// TwinCAT 3 PLC project Untitled1
// ProgramVersion: 3.1.4020.2
// libraries:
//   Tc2_Database, * (Beckhoff Automation GmbH)
//   Tc2_Standard, * (Beckhoff Automation GmbH)
//   Tc2_System, * (Beckhoff Automation GmbH)
//   Tc2_Utilities, * (Beckhoff Automation GmbH)
//   Tc3_Module, * (Beckhoff Automation GmbH)
// project tree:
//   DUTs/ ST_Record.TcDUT
//   GVLs/ GVL.TcGVL
//   / PlcTask.TcTTO
//   POUs/ CheckConnection.TcPOU, DatabaseRecord.TcPOU, DatabaseRetrieve.TcPOU, MAIN.TcPOU
// real-time tasks:
//   TASK PlcTask: cycle T#5ms, priority 20, ADS port 350

CONFIGURATION Untitled1
    RESOURCE PLC ON TwinCAT3
        TASK PlcTask(INTERVAL := T#10ms, PRIORITY := 20);
        PROGRAM MAIN WITH PlcTask : MAIN;
    END_RESOURCE
END_CONFIGURATION

// ---- DUTs/ST_Record.TcDUT
TYPE ST_Record :
STRUCT
	ID: T_ULARGE_INTEGER;
	Timestamp: DT;
	temp1: LREAL;
	temp2: LREAL;
	temp3: LREAL;
	bTest: BYTE;
	sComment: STRING;
END_STRUCT
END_TYPE

// ---- GVLs/GVL.TcGVL

VAR_GLOBAL
	(*------ Variable in the database ------*)
	rTemp1 : REAL;
	rTemp2 : REAL;
	rTemp3 : REAL;
	bToggle : INT;
	sComment: STRING;
	
	tStoreVar : TIME := T#5000MS;
	tRetrieveVar: TIME := T#5000MS;
	stRecord : ST_Record;
	nID: T_ULARGE_INTEGER;
END_VAR

// ---- POUs/MAIN.TcPOU
PROGRAM MAIN
VAR
	randomize : DRAND;
	

END_VAR

(*------ Give random values for temperature ------*)
randomize(Seed:= 1, Num=> );
rTemp1 := randomize.Num * 100;
randomize(Seed:= 1, Num=> );
rTemp2 := randomize.Num * 100;
randomize(Seed:= 1, Num=> );
rTemp3 := randomize.Num * 100;

CheckConnection();
DatabaseRecord();
DatabaseRetrieve();

END_PROGRAM

// ---- POUs/CheckConnection.TcPOU
PROGRAM CheckConnection
VAR
	bInit: BOOL := TRUE;
	fbDBOpen : FB_DBConnectionOpen;
	trigger : R_TRIG;
END_VAR

IF bInit THEN
	fbDBOpen(
		hDBID:= 1, 
		bExecute:= TRUE, 
		tTimeout:= T#5S);
	
	(*------ Throw error if there's any ------*)
	trigger(CLK:= fbDBOpen.bError, Q=> );
	IF trigger.Q THEN
		ADSLOGDINT(msgCtrlMask:= ADSLOG_MSGTYPE_MSGBOX, msgFmtStr:= 'Error connecting to database with error ID: %d', dintArg:=fbDBOpen.nErrID );
		RETURN;
	END_IF
	
	(*------ Continue if there's no problem ------*)
	IF NOT fbDBOpen.bBusy AND NOT fbDBOpen.bError THEN
		fbDBOpen.bExecute := FALSE;
		ADSLOGSTR(msgCtrlMask:= ADSLOG_MSGTYPE_LOG, msgFmtStr:= 'Database connection is good', strArg:= '');
		bInit := FALSE;
	END_IF
END_IF

END_PROGRAM

// ---- POUs/DatabaseRecord.TcPOU
PROGRAM DatabaseRecord
VAR
	tTimeout: TIME := T#5s;
	bExecute: BOOL;
	nState: INT;
	
	fbFormatString: FB_FormatString;
	fbDBRecordSelect: FB_DBRecordArraySelect;
	
	timer: TON := (IN:= TRUE);
END_VAR

(*------ Add data to database every tStoreVar time ------*)
timer(IN:= , PT:= tStoreVar, Q=> , ET=> );

fbDBRecordSelect(
	sNetID:= , 
	hDBID:= 1, 
	pCmdAddr:= , 
	cbCmdSize:= , 
	nStartIndex:= 0, 
	nRecordCount:= 1, 
	pDestAddr:= ADR(nID), 
	cbRecordArraySize:= SIZEOF(nID), 
	bExecute:= , 
	tTimeout:= tTimeout);

fbFormatString(
		sFormat:= 'INSERT INTO [myTable] ([Timestamp],[Temperature1],[Temperature2],[Temperature3], [Status], [Comment]) OUTPUT INSERTED.ID VALUES(CURRENT_TIMESTAMP,%0.5f,%0.5f,%0.5f,%d,$'%s$');',  
		arg1:= F_REAL(rTemp1),
		arg2:= F_REAL(rTemp2),
		arg3:= F_REAL(rTemp3),
		arg4:= F_INT(bToggle),
		arg5:= F_STRING(sComment));
(*
//FORMAT FOR MYSQL 
fbFormatString(
		sFormat:= 'INSERT INTO myTable (Timestamp,Temperature1,Temperature2,Temperature3, Status, Comment) VALUES(CURRENT_TIMESTAMP,%0.5f,%0.5f,%0.5f,%d,$'%s$'); SELECT LAST_INSERT_ID();',  
		arg1:= F_REAL(rTemp1),
		arg2:= F_REAL(rTemp2),
		arg3:= F_REAL(rTemp3),
		arg4:= F_INT(bToggle),
		arg5:= F_STRING(sComment));
*)

(*
//FORMAT FOR SQLite 
fbFormatString(
		sFormat:= 'INSERT INTO [myTable] ([Timestamp],[Temperature1],[Temperature2],[Temperature3], [Status], [Comment]) VALUES(CURRENT_TIMESTAMP,%0.5f,%0.5f,%0.5f,%d,$'%s$'); SELECT LAST_INSERT_ROWID();',  
		arg1:= F_REAL(rTemp1),
		arg2:= F_REAL(rTemp2),
		arg3:= F_REAL(rTemp3),
		arg4:= F_INT(bToggle),
		arg5:= F_STRING(sComment));
*)

CASE nState OF 
	0:
	IF NOT fbFormatString.bError AND fbFormatString.sOut <> '' THEN
		nState := 10;
	END_IF

	10:
	IF timer.Q THEN
		fbDBRecordSelect.pCmdAddr := ADR(fbFormatString.sOut);
		fbDBRecordSelect.cbCmdSize := SIZEOF(fbFormatString.sOut);
		fbDBRecordSelect.bExecute := TRUE;
		timer.IN := FALSE;
		nState := 20;
	END_IF

	20:
	IF NOT fbDBRecordSelect.bBusy AND NOT fbDBRecordSelect.bError THEN
		fbDBRecordSelect.bExecute := FALSE;
		timer.IN := TRUE;
		nState := 0;
	END_IF
END_CASE

END_PROGRAM

// ---- POUs/DatabaseRetrieve.TcPOU
PROGRAM DatabaseRetrieve
VAR
	fbFormatString: FB_FormatString;
	fbDBRecordSelect: FB_DBRecordArraySelect;
	timer : TON := (IN:= TRUE);
	nState: INT;
END_VAR

(*------ Retrive latest data from database every tRetrieveVar time ------*)
timer(IN:= , PT:= tRetrieveVar, Q=> , ET=> );

fbFormatString(
		sFormat:= 'SELECT * FROM [myTable] WHERE ID = %d;',  
		arg1:= F_ULARGE(nId));

fbDBRecordSelect(
	sNetID:= , 
	hDBID:= 1, 
	pCmdAddr:= , 
	cbCmdSize:= , 
	nStartIndex:= 0, 
	nRecordCount:= 1, 
	pDestAddr:= ADR(stRecord), 
	cbRecordArraySize:= SIZEOF(stRecord), 
	bExecute:= , 
	tTimeout:= T#5S, 
	bBusy=> , 
	bError=> , 
	nErrID=> , 
	sSQLState=> , 
	nRecords=> );
	
CASE nState OF
	0:
	IF NOT fbFormatString.bError AND fbFormatString.sOut <> '' THEN
		nState := 10;
	END_IF
	
	10:
	IF timer.Q THEN
		fbDBRecordSelect.pCmdAddr := ADR(fbFormatString.sOut);
		fbDBRecordSelect.cbCmdSize := SIZEOF(fbFormatString.sOut);
		fbDBRecordSelect.bExecute := TRUE;
		timer.IN := FALSE;
		nState := 20;
	END_IF

	20:
	IF NOT fbDBRecordSelect.bBusy AND NOT fbDBRecordSelect.bError THEN
		fbDBRecordSelect.bExecute := FALSE;
		timer.IN := TRUE;
		nState := 0;
	END_IF
END_CASE

END_PROGRAM
